{attribute addProperty BoxType "EL3351-0000-0016"}
{attribute addProperty Id "UnderrangeAT %I*BOOL811OverrangeAT %I*BOOL812ErrorAT %I*BOOL817TxPDO_StateAT %I*BOOL817TxPDO_ToggleAT %I*BOOL819ValueAT %I*DINT32417"}
{attribute addProperty CRC "3965742707"}
{attribute addProperty SizeInBites "72"}
{attribute addProperty SizeInBytes "9"}
TYPE AISupply_Inputs_EC606E73 :
STRUCT
	{attribute addProperty Name "Underrange"}
	Underrange AT %I* : BOOL;
	{attribute addProperty Name "Overrange"}
	Overrange AT %I* : BOOL;
	{attribute addProperty Name "Error"}
	Error AT %I* : BOOL;
	{attribute addProperty Name "TxPDO_State"}
	TxPDO_State AT %I* : BOOL;
	{attribute addProperty Name "TxPDO_Toggle"}
	TxPDO_Toggle AT %I* : BOOL;
	{attribute addProperty Name "Value"}
	Value AT %I* : DINT;
END_STRUCT
END_TYPE

(* stored: Version 1.2.0.0, ProductVersion 3.1.4024.9
   DUT AISupply_Inputs_EC606E73: Id {f3036f48-07ba-4c00-9ec1-91a96f50f9e9} *)
